(* Logix 5000 project; controller EuniceF_ICA6 vendor 1 type 14 code 150 rev 37.11; software revision 37.00 *)

TASK MainTask (continuous, watchdog 500 ms) : MainProgram

MODULES
   Local : vendor 1 type 14 code 150 (Compact 0, rev 37.11)
      Discrete_IO : Embedded (Compact 1, rev 3.1, Output RPI 20 ms)
      Analog_IO : Embedded (Compact 2, rev 1.1, Output RPI 80 ms)
      Counters : Embedded (Compact 3, rev 1.1, Output RPI 20 ms)
END_MODULES

VAR_GLOBAL   (* controller tags *)
   COIL1 : ALIAS FOR Local:1:O.Data.3;
   COIL2 : ALIAS FOR Local:1:O.Data.2;
   HIGH : ALIAS FOR Local:1:I.Data.12;
   LOCK : ALIAS FOR Local:1:O.Data.8;
   RESET : ALIAS FOR Local:1:I.Data.15;
   START : ALIAS FOR Local:1:I.Data.11;
   STOP : ALIAS FOR Local:1:I.Data.8;
   VIB : ALIAS FOR Local:1:I.Data.4;
END_VAR

PROGRAM MainProgram   (* main routine MainRoutine *)

ROUTINE MainRoutine   (* ladder *)
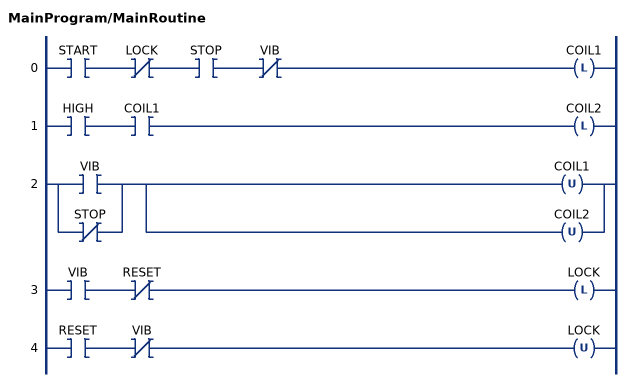
   0: XIC(START)XIO(LOCK)XIC(STOP)XIO(VIB)OTL(COIL1);
   1: XIC(HIGH)XIC(COIL1)OTL(COIL2);
   2: [XIC(VIB) ,XIO(STOP) ][OTU(COIL1) ,OTU(COIL2) ];
   3: XIC(VIB)XIO(RESET)OTL(LOCK);
   4: XIC(RESET)XIO(VIB)OTU(LOCK);
END_ROUTINE
END_PROGRAM
